INTERFACE IOnFail

METHOD CarryOn : BOOL
END_METHOD

METHOD Retry : BOOL
VAR_INPUT
	inFromState : INT;
END_VAR
END_METHOD

METHOD Terminate : BOOL
END_METHOD

END_INTERFACE

(* stored: Version 1.1.0.1, ProductVersion 3.1.4024.9
   Itf IOnFail: Id {64413ada-1c4e-0207-0dd6-42d79018c54f}
   Method CarryOn: Id {9390b52f-558b-082c-1e58-cbe248692714}
   Method Retry: Id {35cbf4b9-b3aa-0f5d-0000-a466366ca062}
   Method Terminate: Id {6bd31019-9b56-0c3f-1fdb-bb53e3d258fc} *)
